LIN {X 0,Y 86.46,Z 826.17,A -85,B 0,C 180,E1 -28946.433,E2 -28946.433} C_VEL
LIN {X 0,Y 94.835,Z 817.694,A -85,B 0,C 180,E1 -28950.553,E2 -28950.553} C_VEL
LIN {X 0,Y 102.155,Z 808.982,A -85,B 0,C 180,E1 -28953.433,E2 -28953.433} C_VEL
LIN {X 0,Y 109.71,Z 798.261,A -85,B 0,C 180,E1 -28955.908,E2 -28955.908} C_VEL
LIN {X 0,Y 115.889,Z 787.44,A -85,B 0,C 180,E1 -28957.648,E2 -28957.648} C_VEL
LIN {X 0,Y 121.383,Z 775.363,A -85,B 0,C 180,E1 -28959.012,E2 -28959.012} C_VEL
LIN {X 0,Y 123.313,Z 770.258,A -85,B 0,C 180,E1 -28959.435,E2 -28959.435} C_VEL
LIN {X 0,Y 124.952,Z 764.764,A -85,B 0,C 180,E1 -28960.101,E2 -28960.101} C_VEL
LIN {X 0,Y 126.471,Z 755.717,A -85,B 0,C 180,E1 -28961.826,E2 -28961.826} C_VEL
LIN {X 0,Y 127.385,Z 746.482,A -85,B 0,C 180,E1 -28963.443,E2 -28963.443} C_VEL
LIN {X 0,Y 127.985,Z 740.687,A -85,B 0,C 180,E1 -28963.94,E2 -28963.94} C_VEL
LIN {X 0,Y 131.877,Z 705.031,A -85,B 0,C 180,E1 -28964.991,E2 -28964.991} C_VEL
LIN {X 0,Y 132.564,Z 694.277,A -85,B 0,C 180,E1 -28966.12,E2 -28966.12} C_VEL
LIN {X 0,Y 131.059,Z 690.593,A -85,B 0,C 180,E1 -28970.158,E2 -28970.158} C_VEL
LIN {X 0,Y 129.868,Z 687.923,A -85,B 0,C 180,E1 -28975.344,E2 -28975.344} C_VEL
LIN {X 0,Y 129.584,Z 687.04,A -85,B 0,C 180,E1 -28978.446,E2 -28978.446} C_VEL
LIN {X 0,Y 129.581,Z 688.078,A -85,B 0,C 180,E1 -28983.109,E2 -28983.109} C_VEL
LIN {X 0,Y 130.12,Z 690.292,A -85,B 0,C 180,E1 -28987.175,E2 -28987.175} C_VEL
LIN {X 0,Y 131.254,Z 694.381,A -85,B 0,C 180,E1 -28991.584,E2 -28991.584} C_VEL
LIN {X 0,Y 132.585,Z 699.79,A -85,B 0,C 180,E1 -28995.273,E2 -28995.273} C_VEL
LIN {X 0,Y 129.78,Z 725.663,A -85,B 0,C 180,E1 -28996.051,E2 -28996.051} C_VEL
LIN {X 0,Y 127.305,Z 745.814,A -85,B 0,C 180,E1 -28996.653,E2 -28996.653} C_VEL
LIN {X 0,Y 124.21,Z 759.298,A -85,B 0,C 180,E1 -28997.284,E2 -28997.284} C_VEL
LIN {X 0,Y 120.227,Z 771.36,A -85,B 0,C 180,E1 -28998.205,E2 -28998.205} C_VEL
LIN {X 0,Y 115.453,Z 782.235,A -85,B 0,C 180,E1 -28999.34,E2 -28999.34} C_VEL
LIN {X 0,Y 109.154,Z 793.548,A -85,B 0,C 180,E1 -29000.991,E2 -29000.991} C_VEL
LIN {X 0,Y 102.148,Z 803.754,A -85,B 0,C 180,E1 -29003.034,E2 -29003.034} C_VEL
LIN {X 0,Y 95.328,Z 812.1,A -85,B 0,C 180,E1 -29005.422,E2 -29005.422} C_VEL
LIN {X 0,Y 87.086,Z 820.636,A -85,B 0,C 180,E1 -29008.961,E2 -29008.961} C_VEL
LIN {X 0,Y 78.237,Z 828.356,A -85,B 0,C 180,E1 -29013.8,E2 -29013.8} C_VEL
LIN {X 0,Y 69.093,Z 834.993,A -85,B 0,C 180,E1 -29020.274,E2 -29020.274} C_VEL
LIN {X 0,Y 62.144,Z 839.341,A -85,B 0,C 180,E1 -29027.262,E2 -29027.262} C_VEL
LIN {X 0,Y 58.152,Z 841.624,A -85,B 0,C 180,E1 -29032.817,E2 -29032.817} C_VEL
LIN {X 0,Y 54.742,Z 843.484,A -85,B 0,C 180,E1 -29039.094,E2 -29039.094} C_VEL
LIN {X 0,Y 52.001,Z 844.896,A -85,B 0,C 180,E1 -29046.074,E2 -29046.074} C_VEL
LIN {X 0,Y 48.874,Z 846.492,A -85,B 0,C 180,E1 -29061.726,E2 -29061.726} C_VEL
LIN {X 0,Y 48.51,Z 846.718,A -85,B 0,C 180,E1 -29069.993,E2 -29069.993} C_VEL
LIN {X 0,Y 48.829,Z 846.519,A -85,B 0,C 180,E1 -29078.268,E2 -29078.268} C_VEL
LIN {X 0,Y 50.012,Z 845.929,A -85,B 0,C 180,E1 -29086.316,E2 -29086.316} C_VEL
LIN {X 0,Y 51.995,Z 844.956,A -85,B 0,C 180,E1 -29093.915,E2 -29093.915} C_VEL
LIN {X 0,Y 54.73,Z 843.578,A -85,B 0,C 180,E1 -29100.9,E2 -29100.9} C_VEL
LIN {X 0,Y 60.066,Z 840.685,A -85,B 0,C 180,E1 -29110.047,E2 -29110.047} C_VEL
LIN {X 0,Y 66.591,Z 836.748,A -85,B 0,C 180,E1 -29117.619,E2 -29117.619} C_VEL
LIN {X 0,Y 74.148,Z 831.639,A -85,B 0,C 180,E1 -29123.665,E2 -29123.665} C_VEL
LIN {X 0,Y 82.281,Z 825.202,A -85,B 0,C 180,E1 -29128.656,E2 -29128.656} C_VEL
LIN {X 0,Y 84.018,Z 823.562,A -85,B 0,C 180,E1 -29129.874,E2 -29129.874} C_VEL
LIN {X 0,Y 78.219,Z 822.134,A -85,B 0,C 180,E1 -29144.362,E2 -29144.362} C_VEL
LIN {X 0,Y 78.822,Z 819.937,A -85,B 0,C 180,E1 -29160,E2 -29160} C_VEL
LIN {X 0,Y 85.752,Z 816.801,A -85,B 0,C 180,E1 -29174.233,E2 -29174.233} C_VEL
LIN {X 0,Y 94.96,Z 813.582,A -85,B 0,C 180,E1 -29183.594,E2 -29183.594} C_VEL
LIN {X 0,Y 94.804,Z 814.301,A -85,B 0,C 180,E1 -29184.407,E2 -29184.407} C_VEL
LIN {X 0,Y 87.113,Z 822.244,A -85,B 0,C 180,E1 -29187.456,E2 -29187.456} C_VEL
LIN {X 0,Y 78.562,Z 829.753,A -85,B 0,C 180,E1 -29191.814,E2 -29191.814} C_VEL
LIN {X 0,Y 70.637,Z 835.789,A -85,B 0,C 180,E1 -29197.263,E2 -29197.263} C_VEL
LIN {X 0,Y 63.363,Z 840.558,A -85,B 0,C 180,E1 -29203.875,E2 -29203.875} C_VEL
LIN {X 0,Y 57.146,Z 844.205,A -85,B 0,C 180,E1 -29212.062,E2 -29212.062} C_VEL
LIN {X 0,Y 53.773,Z 846.089,A -85,B 0,C 180,E1 -29218.488,E2 -29218.488} C_VEL
LIN {X 0,Y 51.191,Z 847.509,A -85,B 0,C 180,E1 -29225.685,E2 -29225.685} C_VEL
LIN {X 0,Y 48.553,Z 849.137,A -85,B 0,C 180,E1 -29241.684,E2 -29241.684} C_VEL
LIN {X 0,Y 48.502,Z 849.357,A -85,B 0,C 180,E1 -29250.007,E2 -29250.007} C_VEL
LIN {X 0,Y 48.555,Z 849.116,A -85,B 0,C 180,E1 -29258.329,E2 -29258.329} C_VEL
LIN {X 0,Y 51.19,Z 847.46,A -85,B 0,C 180,E1 -29274.329,E2 -29274.329} C_VEL
LIN {X 0,Y 53.765,Z 846.011,A -85,B 0,C 180,E1 -29281.531,E2 -29281.531} C_VEL
LIN {X 0,Y 59.08,Z 843.026,A -85,B 0,C 180,E1 -29290.871,E2 -29290.871} C_VEL
LIN {X 0,Y 65.662,Z 838.985,A -85,B 0,C 180,E1 -29298.53,E2 -29298.53} C_VEL
LIN {X 0,Y 73.734,Z 833.34,A -85,B 0,C 180,E1 -29305.118,E2 -29305.118} C_VEL
LIN {X 0,Y 82.731,Z 825.978,A -85,B 0,C 180,E1 -29310.551,E2 -29310.551} C_VEL
LIN {X 0,Y 91.551,Z 817.503,A -85,B 0,C 180,E1 -29314.429,E2 -29314.429} C_VEL
LIN {X 0,Y 99.175,Z 808.792,A -85,B 0,C 180,E1 -29317.114,E2 -29317.114} C_VEL
LIN {X 0,Y 107.013,Z 798.075,A -85,B 0,C 180,E1 -29319.374,E2 -29319.374} C_VEL
LIN {X 0,Y 113.383,Z 787.257,A -85,B 0,C 180,E1 -29320.962,E2 -29320.962} C_VEL
LIN {X 0,Y 119.028,Z 775.186,A -85,B 0,C 180,E1 -29322.201,E2 -29322.201} C_VEL
LIN {X 0,Y 123.519,Z 762.455,A -85,B 0,C 180,E1 -29323.064,E2 -29323.064} C_VEL
LIN {X 0,Y 126.616,Z 749.727,A -85,B 0,C 180,E1 -29323.597,E2 -29323.597} C_VEL
LIN {X 0,Y 127.985,Z 740.687,A -85,B 0,C 180,E1 -29323.94,E2 -29323.94} C_VEL
LIN {X 0,Y 128.477,Z 734.891,A -85,B 0,C 180,E1 -29324.411,E2 -29324.411} C_VEL
LIN {X 0,Y 129.14,Z 716.204,A -85,B 0,C 180,E1 -29327.354,E2 -29327.354} C_VEL
LIN {X 0,Y 129.631,Z 710.401,A -85,B 0,C 180,E1 -29327.808,E2 -29327.808} C_VEL
LIN {X 0,Y 130.259,Z 704.044,A -85,B 0,C 180,E1 -29328.159,E2 -29328.159} C_VEL
LIN {X 0,Y 130.607,Z 699.268,A -85,B 0,C 180,E1 -29328.692,E2 -29328.692} C_VEL
LIN {X 0,Y 129.778,Z 697.071,A -85,B 0,C 180,E1 -29331.436,E2 -29331.436} C_VEL
LIN {X 0,Y 128.943,Z 694.914,A -85,B 0,C 180,E1 -29335.702,E2 -29335.702} C_VEL
LIN {X 0,Y 128.714,Z 694.127,A -85,B 0,C 180,E1 -29338.436,E2 -29338.436} C_VEL
LIN {X 0,Y 128.669,Z 695.009,A -85,B 0,C 180,E1 -29342.563,E2 -29342.563} C_VEL
LIN {X 0,Y 129.078,Z 697.136,A -85,B 0,C 180,E1 -29346.44,E2 -29346.44} C_VEL
LIN {X 0,Y 129.961,Z 700.948,A -85,B 0,C 180,E1 -29350.516,E2 -29350.516} C_VEL
LIN {X 0,Y 130.496,Z 703.71,A -85,B 0,C 180,E1 -29352.441,E2 -29352.441} C_VEL
LIN {X 0,Y 125.582,Z 745.27,A -85,B 0,C 180,E1 -29353.527,E2 -29353.527} C_VEL
LIN {X 0,Y 122.71,Z 758.014,A -85,B 0,C 180,E1 -29354.047,E2 -29354.047} C_VEL
LIN {X 0,Y 118.615,Z 770.448,A -85,B 0,C 180,E1 -29354.859,E2 -29354.859} C_VEL
LIN {X 0,Y 113.301,Z 782.417,A -85,B 0,C 180,E1 -29355.952,E2 -29355.952} C_VEL
LIN {X 0,Y 106.824,Z 793.734,A -85,B 0,C 180,E1 -29357.445,E2 -29357.445} C_VEL
LIN {X 0,Y 99.59,Z 803.943,A -85,B 0,C 180,E1 -29359.282,E2 -29359.282} C_VEL
LIN {X 0,Y 92.501,Z 812.291,A -85,B 0,C 180,E1 -29361.444,E2 -29361.444} C_VEL
LIN {X 0,Y 84.831,Z 819.972,A -85,B 0,C 180,E1 -29364.304,E2 -29364.304} C_VEL
LIN {X 0,Y 75.941,Z 827.453,A -85,B 0,C 180,E1 -29368.449,E2 -29368.449} C_VEL
LIN {X 0,Y 67.442,Z 833.459,A -85,B 0,C 180,E1 -29373.516,E2 -29373.516} C_VEL
LIN {X 0,Y 59.557,Z 838.201,A -85,B 0,C 180,E1 -29379.904,E2 -29379.904} C_VEL
LIN {X 0,Y 52.675,Z 841.817,A -85,B 0,C 180,E1 -29388.148,E2 -29388.148} C_VEL
LIN {X 0,Y 48.78,Z 843.677,A -85,B 0,C 180,E1 -29394.801,E2 -29394.801} C_VEL
LIN {X 0,Y 45.601,Z 845.089,A -85,B 0,C 180,E1 -29402.453,E2 -29402.453} C_VEL
LIN {X 0,Y 41.877,Z 846.685,A -85,B 0,C 180,E1 -29420.331,E2 -29420.331} C_VEL
LIN {X 0,Y 41.428,Z 846.911,A -85,B 0,C 180,E1 -29429.992,E2 -29429.992} C_VEL
LIN {X 0,Y 41.826,Z 846.712,A -85,B 0,C 180,E1 -29439.665,E2 -29439.665} C_VEL
LIN {X 0,Y 45.594,Z 845.149,A -85,B 0,C 180,E1 -29457.535,E2 -29457.535} C_VEL
LIN {X 0,Y 48.767,Z 843.771,A -85,B 0,C 180,E1 -29465.193,E2 -29465.193} C_VEL
LIN {X 0,Y 54.802,Z 840.878,A -85,B 0,C 180,E1 -29474.848,E2 -29474.848} C_VEL
LIN {X 0,Y 62.034,Z 836.939,A -85,B 0,C 180,E1 -29482.462,E2 -29482.462} C_VEL
LIN {X 0,Y 70.178,Z 831.829,A -85,B 0,C 180,E1 -29488.336,E2 -29488.336} C_VEL
LIN {X 0,Y 75.329,Z 828.108,A -85,B 0,C 180,E1 -29491.331,E2 -29491.331} C_VEL
LIN {X 0,Y 76.161,Z 827.21,A -85,B 0,C 180,E1 -29492.522,E2 -29492.522} C_VEL
LIN {X 0,Y 71.978,Z 825.743,A -85,B 0,C 180,E1 -29508.738,E2 -29508.738} C_VEL
LIN {X 0,Y 74.833,Z 823.501,A -85,B 0,C 180,E1 -29525.389,E2 -29525.389} C_VEL
LIN {X 0,Y 85.395,Z 819.982,A -85,B 0,C 180,E1 -29540.986,E2 -29540.986} C_VEL
LIN {X 0,Y 86.136,Z 819.753,A -85,B 0,C 180,E1 -29541.678,E2 -29541.678} C_VEL
LIN {X 0,Y 84.717,Z 821.456,A -85,B 0,C 180,E1 -29542.901,E2 -29542.901} C_VEL
LIN {X 0,Y 75.043,Z 829.563,A -85,B 0,C 180,E1 -29547.176,E2 -29547.176} C_VEL
LIN {X 0,Y 66.551,Z 835.598,A -85,B 0,C 180,E1 -29552.357,E2 -29552.357} C_VEL
LIN {X 0,Y 58.639,Z 840.366,A -85,B 0,C 180,E1 -29558.837,E2 -29558.837} C_VEL
LIN {X 0,Y 51.721,Z 844.013,A -85,B 0,C 180,E1 -29567.212,E2 -29567.212} C_VEL
LIN {X 0,Y 47.83,Z 845.896,A -85,B 0,C 180,E1 -29574.012,E2 -29574.012} C_VEL
LIN {X 0,Y 44.782,Z 847.316,A -85,B 0,C 180,E1 -29581.922,E2 -29581.922} C_VEL
LIN {X 0,Y 41.528,Z 848.944,A -85,B 0,C 180,E1 -29600.265,E2 -29600.265} C_VEL
LIN {X 0,Y 41.412,Z 849.164,A -85,B 0,C 180,E1 -29610.008,E2 -29610.008} C_VEL
LIN {X 0,Y 41.529,Z 848.923,A -85,B 0,C 180,E1 -29619.751,E2 -29619.751} C_VEL
LIN {X 0,Y 44.782,Z 847.266,A -85,B 0,C 180,E1 -29638.095,E2 -29638.095} C_VEL
LIN {X 0,Y 47.823,Z 845.817,A -85,B 0,C 180,E1 -29646.011,E2 -29646.011} C_VEL
LIN {X 0,Y 53.889,Z 842.832,A -85,B 0,C 180,E1 -29655.839,E2 -29655.839} C_VEL
LIN {X 0,Y 61.185,Z 838.791,A -85,B 0,C 180,E1 -29663.526,E2 -29663.526} C_VEL
LIN {X 0,Y 70.675,Z 832.593,A -85,B 0,C 180,E1 -29670.406,E2 -29670.406} C_VEL
LIN {X 0,Y 79.474,Z 825.785,A -85,B 0,C 180,E1 -29675.024,E2 -29675.024} C_VEL
LIN {X 0,Y 88.709,Z 817.312,A -85,B 0,C 180,E1 -29678.583,E2 -29678.583} C_VEL
LIN {X 0,Y 96.629,Z 808.603,A -85,B 0,C 180,E1 -29681.007,E2 -29681.007} C_VEL
LIN {X 0,Y 104.727,Z 797.888,A -85,B 0,C 180,E1 -29683.004,E2 -29683.004} C_VEL
LIN {X 0,Y 111.273,Z 787.074,A -85,B 0,C 180,E1 -29684.414,E2 -29684.414} C_VEL
LIN {X 0,Y 117.056,Z 775.009,A -85,B 0,C 180,E1 -29685.506,E2 -29685.506} C_VEL
LIN {X 0,Y 121.644,Z 762.29,A -85,B 0,C 180,E1 -29686.258,E2 -29686.258} C_VEL
LIN {X 0,Y 124.881,Z 749.158,A -85,B 0,C 180,E1 -29686.738,E2 -29686.738} C_VEL
LIN {X 0,Y 127.205,Z 731.857,A -85,B 0,C 180,E1 -29687.264,E2 -29687.264} C_VEL
LIN {X 0,Y 129.631,Z 710.401,A -85,B 0,C 180,E1 -29687.808,E2 -29687.808} C_VEL
LIN {X 0,Y 129.736,Z 707.831,A -85,B 0,C 180,E1 -29688.259,E2 -29688.259} C_VEL
LIN {X 0,Y 129.517,Z 705.447,A -85,B 0,C 180,E1 -29689.408,E2 -29689.408} C_VEL
LIN {X 0,Y 129.091,Z 703.798,A -85,B 0,C 180,E1 -29691.014,E2 -29691.014} C_VEL
LIN {X 0,Y 128.425,Z 702.558,A -85,B 0,C 180,E1 -29693.701,E2 -29693.701} C_VEL
LIN {X 0,Y 127.977,Z 701.798,A -85,B 0,C 180,E1 -29696.453,E2 -29696.453} C_VEL
LIN {X 0,Y 127.848,Z 701.182,A -85,B 0,C 180,E1 -29698.425,E2 -29698.425} C_VEL
LIN {X 0,Y 127.78,Z 702.05,A -85,B 0,C 180,E1 -29702.295,E2 -29702.295} C_VEL
LIN {X 0,Y 128.083,Z 704.162,A -85,B 0,C 180,E1 -29705.905,E2 -29705.905} C_VEL
LIN {X 0,Y 128.712,Z 707.544,A -85,B 0,C 180,E1 -29709.428,E2 -29709.428} C_VEL
LIN {X 0,Y 124.023,Z 745.927,A -85,B 0,C 180,E1 -29710.359,E2 -29710.359} C_VEL
LIN {X 0,Y 120.97,Z 758.904,A -85,B 0,C 180,E1 -29710.815,E2 -29710.815} C_VEL
LIN {X 0,Y 116.583,Z 771.711,A -85,B 0,C 180,E1 -29711.582,E2 -29711.582} C_VEL
LIN {X 0,Y 111.562,Z 782.599,A -85,B 0,C 180,E1 -29712.451,E2 -29712.451} C_VEL
LIN {X 0,Y 104.92,Z 793.92,A -85,B 0,C 180,E1 -29713.756,E2 -29713.756} C_VEL
LIN {X 0,Y 97.481,Z 804.13,A -85,B 0,C 180,E1 -29715.35,E2 -29715.35} C_VEL
LIN {X 0,Y 90.145,Z 812.481,A -85,B 0,C 180,E1 -29717.234,E2 -29717.234} C_VEL
LIN {X 0,Y 82.166,Z 820.163,A -85,B 0,C 180,E1 -29719.791,E2 -29719.791} C_VEL
LIN {X 0,Y 72.817,Z 827.646,A -85,B 0,C 180,E1 -29723.514,E2 -29723.514} C_VEL
LIN {X 0,Y 63.8,Z 833.652,A -85,B 0,C 180,E1 -29728.197,E2 -29728.197} C_VEL
LIN {X 0,Y 55.274,Z 838.394,A -85,B 0,C 180,E1 -29734.254,E2 -29734.254} C_VEL
LIN {X 0,Y 47.629,Z 842.01,A -85,B 0,C 180,E1 -29742.448,E2 -29742.448} C_VEL
LIN {X 0,Y 43.172,Z 843.871,A -85,B 0,C 180,E1 -29749.362,E2 -29749.362} C_VEL
LIN {X 0,Y 39.449,Z 845.282,A -85,B 0,C 180,E1 -29757.683,E2 -29757.683} C_VEL
LIN {X 0,Y 34.892,Z 846.878,A -85,B 0,C 180,E1 -29778.37,E2 -29778.37} C_VEL
LIN {X 0,Y 34.331,Z 847.104,A -85,B 0,C 180,E1 -29789.99,E2 -29789.99} C_VEL
LIN {X 0,Y 34.843,Z 846.905,A -85,B 0,C 180,E1 -29801.627,E2 -29801.627} C_VEL
LIN {X 0,Y 39.441,Z 845.341,A -85,B 0,C 180,E1 -29822.304,E2 -29822.304} C_VEL
LIN {X 0,Y 43.159,Z 843.963,A -85,B 0,C 180,E1 -29830.634,E2 -29830.634} C_VEL
LIN {X 0,Y 50.007,Z 841.07,A -85,B 0,C 180,E1 -29840.61,E2 -29840.61} C_VEL
LIN {X 0,Y 57.989,Z 837.129,A -85,B 0,C 180,E1 -29848.022,E2 -29848.022} C_VEL
LIN {X 0,Y 66.375,Z 832.252,A -85,B 0,C 180,E1 -29853.334,E2 -29853.334} C_VEL
LIN {X 0,Y 68.453,Z 830.543,A -85,B 0,C 180,E1 -29855.752,E2 -29855.752} C_VEL
LIN {X 0,Y 66.127,Z 829.096,A -85,B 0,C 180,E1 -29873.899,E2 -29873.899} C_VEL
LIN {X 0,Y 71.877,Z 826.736,A -85,B 0,C 180,E1 -29892.128,E2 -29892.128} C_VEL
LIN {X 0,Y 76.932,Z 825.362,A -85,B 0,C 180,E1 -29899.207,E2 -29899.207} C_VEL
LIN {X 0,Y 75.181,Z 827.044,A -85,B 0,C 180,E1 -29900.816,E2 -29900.816} C_VEL
LIN {X 0,Y 65.075,Z 834.136,A -85,B 0,C 180,E1 -29905.594,E2 -29905.594} C_VEL
LIN {X 0,Y 57.252,Z 838.74,A -85,B 0,C 180,E1 -29910.776,E2 -29910.776} C_VEL
LIN {X 0,Y 49.201,Z 842.747,A -85,B 0,C 180,E1 -29918.233,E2 -29918.233} C_VEL
LIN {X 0,Y 42.262,Z 845.703,A -85,B 0,C 180,E1 -29928.316,E2 -29928.316} C_VEL
LIN {X 0,Y 38.637,Z 847.122,A -85,B 0,C 180,E1 -29936.939,E2 -29936.939} C_VEL
LIN {X 0,Y 34.531,Z 848.75,A -85,B 0,C 180,E1 -29958.267,E2 -29958.267} C_VEL
LIN {X 0,Y 34.307,Z 848.971,A -85,B 0,C 180,E1 -29970.01,E2 -29970.01} C_VEL
LIN {X 0,Y 34.533,Z 848.729,A -85,B 0,C 180,E1 -29981.752,E2 -29981.752} C_VEL
LIN {X 0,Y 38.638,Z 847.071,A -85,B 0,C 180,E1 -30003.081,E2 -30003.081} C_VEL
LIN {X 0,Y 42.257,Z 845.622,A -85,B 0,C 180,E1 -30011.712,E2 -30011.712} C_VEL
LIN {X 0,Y 49.189,Z 842.638,A -85,B 0,C 180,E1 -30021.807,E2 -30021.807} C_VEL
LIN {X 0,Y 57.243,Z 838.598,A -85,B 0,C 180,E1 -30029.261,E2 -30029.261} C_VEL
LIN {X 0,Y 66.193,Z 833.231,A -85,B 0,C 180,E1 -30035.014,E2 -30035.014} C_VEL
LIN {X 0,Y 75.158,Z 826.814,A -85,B 0,C 180,E1 -30039.253,E2 -30039.253} C_VEL
LIN {X 0,Y 84.746,Z 818.677,A -85,B 0,C 180,E1 -30042.507,E2 -30042.507} C_VEL
LIN {X 0,Y 92.912,Z 810.333,A -85,B 0,C 180,E1 -30044.683,E2 -30044.683} C_VEL
LIN {X 0,Y 101.204,Z 800.015,A -85,B 0,C 180,E1 -30046.472,E2 -30046.472} C_VEL
LIN {X 0,Y 108.738,Z 788.416,A -85,B 0,C 180,E1 -30047.85,E2 -30047.85} C_VEL
LIN {X 0,Y 114.635,Z 776.765,A -85,B 0,C 180,E1 -30048.8,E2 -30048.8} C_VEL
LIN {X 0,Y 119.306,Z 764.743,A -85,B 0,C 180,E1 -30049.436,E2 -30049.436} C_VEL
LIN {X 0,Y 122.867,Z 751.939,A -85,B 0,C 180,E1 -30049.855,E2 -30049.855} C_VEL
LIN {X 0,Y 125.197,Z 737.19,A -85,B 0,C 180,E1 -30050.305,E2 -30050.305} C_VEL
LIN {X 0,Y 128.68,Z 707.099,A -85,B 0,C 180,E1 -30051.015,E2 -30051.015} C_VEL
LIN {X 0,Y 128.913,Z 704.421,A -85,B 0,C 180,E1 -30051.298,E2 -30051.298} C_VEL
LIN {X 0,Y 128.031,Z 701.961,A -85,B 0,C 180,E1 -30055.967,E2 -30055.967} C_VEL
LIN {X 0,Y 127.977,Z 701.798,A -85,B 0,C 180,E1 -30056.453,E2 -30056.453} C_VEL
LIN {X 0,Y 127.743,Z 702.175,A -85,B 0,C 180,E1 -30058.174,E2 -30058.174} C_VEL
LIN {X 0,Y 127.477,Z 703.765,A -85,B 0,C 180,E1 -30059.798,E2 -30059.798} C_VEL
LIN {X 0,Y 127.018,Z 710.164,A -85,B 0,C 180,E1 -30064.224,E2 -30064.224} C_VEL
LIN {X 0,Y 127.072,Z 710.961,A -85,B 0,C 180,E1 -30065.091,E2 -30065.091} C_VEL
LIN {X 0,Y 127.212,Z 712.043,A -85,B 0,C 180,E1 -30066.344,E2 -30066.344} C_VEL
LIN {X 0,Y 123.014,Z 745.705,A -85,B 0,C 180,E1 -30067.104,E2 -30067.104} C_VEL
LIN {X 0,Y 119.845,Z 759.068,A -85,B 0,C 180,E1 -30067.494,E2 -30067.494} C_VEL
LIN {X 0,Y 115.371,Z 771.886,A -85,B 0,C 180,E1 -30068.139,E2 -30068.139} C_VEL
LIN {X 0,Y 110.25,Z 782.781,A -85,B 0,C 180,E1 -30068.848,E2 -30068.848} C_VEL
LIN {X 0,Y 103.464,Z 794.105,A -85,B 0,C 180,E1 -30069.943,E2 -30069.943} C_VEL
LIN {X 0,Y 95.848,Z 804.319,A -85,B 0,C 180,E1 -30071.257,E2 -30071.257} C_VEL
LIN {X 0,Y 88.303,Z 812.671,A -85,B 0,C 180,E1 -30072.833,E2 -30072.833} C_VEL
LIN {X 0,Y 78.631,Z 821.506,A -85,B 0,C 180,E1 -30075.402,E2 -30075.402} C_VEL
LIN {X 0,Y 68.694,Z 828.935,A -85,B 0,C 180,E1 -30078.839,E2 -30078.839} C_VEL
LIN {X 0,Y 57.668,Z 835.571,A -85,B 0,C 180,E1 -30083.919,E2 -30083.919} C_VEL
LIN {X 0,Y 48.67,Z 839.922,A -85,B 0,C 180,E1 -30089.944,E2 -30089.944} C_VEL
LIN {X 0,Y 43.149,Z 842.204,A -85,B 0,C 180,E1 -30095.462,E2 -30095.462} C_VEL
LIN {X 0,Y 38.072,Z 844.064,A -85,B 0,C 180,E1 -30102.394,E2 -30102.394} C_VEL
LIN {X 0,Y 33.651,Z 845.476,A -85,B 0,C 180,E1 -30111.192,E2 -30111.192} C_VEL
LIN {X 0,Y 27.969,Z 847.072,A -85,B 0,C 180,E1 -30135.435,E2 -30135.435} C_VEL
LIN {X 0,Y 27.248,Z 847.297,A -85,B 0,C 180,E1 -30149.988,E2 -30149.988} C_VEL
LIN {X 0,Y 27.93,Z 847.097,A -85,B 0,C 180,E1 -30164.561,E2 -30164.561} C_VEL
LIN {X 0,Y 30.175,Z 846.507,A -85,B 0,C 180,E1 -30177.75,E2 -30177.75} C_VEL
LIN {X 0,Y 33.641,Z 845.534,A -85,B 0,C 180,E1 -30188.796,E2 -30188.796} C_VEL
LIN {X 0,Y 38.056,Z 844.155,A -85,B 0,C 180,E1 -30197.607,E2 -30197.607} C_VEL
LIN {X 0,Y 45.824,Z 841.261,A -85,B 0,C 180,E1 -30207.5,E2 -30207.5} C_VEL
LIN {X 0,Y 54.568,Z 837.319,A -85,B 0,C 180,E1 -30214.347,E2 -30214.347} C_VEL
LIN {X 0,Y 60.729,Z 834.03,A -85,B 0,C 180,E1 -30217.775,E2 -30217.775} C_VEL
LIN {X 0,Y 60.894,Z 833.617,A -85,B 0,C 180,E1 -30219.742,E2 -30219.742} C_VEL
LIN {X 0,Y 60.88,Z 832.161,A -85,B 0,C 180,E1 -30240,E2 -30240} C_VEL
LIN {X 0,Y 67.672,Z 830.257,A -85,B 0,C 180,E1 -30256.159,E2 -30256.159} C_VEL
LIN {X 0,Y 66.467,Z 831.366,A -85,B 0,C 180,E1 -30257.913,E2 -30257.913} C_VEL
LIN {X 0,Y 57.026,Z 836.945,A -85,B 0,C 180,E1 -30262.453,E2 -30262.453} C_VEL
LIN {X 0,Y 47.983,Z 841.319,A -85,B 0,C 180,E1 -30268.518,E2 -30268.518} C_VEL
LIN {X 0,Y 42.382,Z 843.628,A -85,B 0,C 180,E1 -30274.006,E2 -30274.006} C_VEL
LIN {X 0,Y 37.237,Z 845.509,A -85,B 0,C 180,E1 -30280.993,E2 -30280.993} C_VEL
LIN {X 0,Y 32.898,Z 846.929,A -85,B 0,C 180,E1 -30290.156,E2 -30290.156} C_VEL
LIN {X 0,Y 27.612,Z 848.557,A -85,B 0,C 180,E1 -30315.267,E2 -30315.267} C_VEL
LIN {X 0,Y 27.218,Z 848.778,A -85,B 0,C 180,E1 -30330.012,E2 -30330.012} C_VEL
LIN {X 0,Y 27.614,Z 848.535,A -85,B 0,C 180,E1 -30344.757,E2 -30344.757} C_VEL
LIN {X 0,Y 32.9,Z 846.878,A -85,B 0,C 180,E1 -30369.868,E2 -30369.868} C_VEL
LIN {X 0,Y 37.231,Z 845.428,A -85,B 0,C 180,E1 -30379.043,E2 -30379.043} C_VEL
LIN {X 0,Y 45.13,Z 842.443,A -85,B 0,C 180,E1 -30388.94,E2 -30388.94} C_VEL
LIN {X 0,Y 53.954,Z 838.404,A -85,B 0,C 180,E1 -30395.771,E2 -30395.771} C_VEL
LIN {X 0,Y 64.709,Z 832.281,A -85,B 0,C 180,E1 -30401.386,E2 -30401.386} C_VEL
LIN {X 0,Y 74.582,Z 825.4,A -85,B 0,C 180,E1 -30405.003,E2 -30405.003} C_VEL
LIN {X 0,Y 84.554,Z 816.93,A -85,B 0,C 180,E1 -30407.605,E2 -30407.605} C_VEL
LIN {X 0,Y 92.976,Z 808.224,A -85,B 0,C 180,E1 -30409.33,E2 -30409.33} C_VEL
LIN {X 0,Y 101.492,Z 797.516,A -85,B 0,C 180,E1 -30410.685,E2 -30410.685} C_VEL
LIN {X 0,Y 108.329,Z 786.709,A -85,B 0,C 180,E1 -30411.653,E2 -30411.653} C_VEL
LIN {X 0,Y 114.332,Z 774.654,A -85,B 0,C 180,E1 -30412.41,E2 -30412.41} C_VEL
LIN {X 0,Y 119.074,Z 761.958,A -85,B 0,C 180,E1 -30412.906,E2 -30412.906} C_VEL
LIN {X 0,Y 122.47,Z 748.533,A -85,B 0,C 180,E1 -30413.24,E2 -30413.24} C_VEL
LIN {X 0,Y 124.846,Z 731.669,A -85,B 0,C 180,E1 -30413.625,E2 -30413.625} C_VEL
LIN {X 0,Y 127.405,Z 709.97,A -85,B 0,C 180,E1 -30414.133,E2 -30414.133} C_VEL
LIN {X 0,Y 126.974,Z 708.299,A -85,B 0,C 180,E1 -30418.414,E2 -30418.414} C_VEL
LIN {X 0,Y 126.884,Z 708.928,A -85,B 0,C 180,E1 -30421.587,E2 -30421.587} C_VEL
LIN {X 0,Y 127.039,Z 710.648,A -85,B 0,C 180,E1 -30424.701,E2 -30424.701} C_VEL
LIN {X 0,Y 127.072,Z 710.961,A -85,B 0,C 180,E1 -30425.091,E2 -30425.091} C_VEL
LIN {X 0,Y 127.037,Z 712.212,A -85,B 0,C 180,E1 -30425.671,E2 -30425.671} C_VEL
LIN {X 0,Y 126.791,Z 714.634,A -85,B 0,C 180,E1 -30425.91,E2 -30425.91} C_VEL
LIN {X 0,Y 126.263,Z 718.398,A -85,B 0,C 180,E1 -30425.62,E2 -30425.62} C_VEL
LIN {X 0,Y 124.887,Z 727.073,A -85,B 0,C 180,E1 -30423.906,E2 -30423.906} C_VEL
LIN {X 0,Y 124.355,Z 730.999,A -85,B 0,C 180,E1 -30423.547,E2 -30423.547} C_VEL
LIN {X 0,Y 124.256,Z 731.801,A -85,B 0,C 180,E1 -30423.548,E2 -30423.548} C_VEL
LIN {X 0,Y 121.901,Z 748.043,A -85,B 0,C 180,E1 -30423.868,E2 -30423.868} C_VEL
LIN {X 0,Y 118.476,Z 761.412,A -85,B 0,C 180,E1 -30424.169,E2 -30424.169} C_VEL
LIN {X 0,Y 114.584,Z 772.061,A -85,B 0,C 180,E1 -30424.634,E2 -30424.634} C_VEL
LIN {X 0,Y 109.384,Z 782.963,A -85,B 0,C 180,E1 -30425.175,E2 -30425.175} C_VEL
LIN {X 0,Y 102.479,Z 794.29,A -85,B 0,C 180,E1 -30426.038,E2 -30426.038} C_VEL
LIN {X 0,Y 94.719,Z 804.507,A -85,B 0,C 180,E1 -30427.045,E2 -30427.045} C_VEL
LIN {X 0,Y 87.004,Z 812.861,A -85,B 0,C 180,E1 -30428.276,E2 -30428.276} C_VEL
LIN {X 0,Y 78.498,Z 820.547,A -85,B 0,C 180,E1 -30429.971,E2 -30429.971} C_VEL
LIN {X 0,Y 68.401,Z 828.031,A -85,B 0,C 180,E1 -30432.535,E2 -30432.535} C_VEL
LIN {X 0,Y 58.452,Z 834.037,A -85,B 0,C 180,E1 -30435.854,E2 -30435.854} C_VEL
LIN {X 0,Y 48.706,Z 838.781,A -85,B 0,C 180,E1 -30440.278,E2 -30440.278} C_VEL
LIN {X 0,Y 39.453,Z 842.398,A -85,B 0,C 180,E1 -30447.025,E2 -30447.025} C_VEL
LIN {X 0,Y 33.693,Z 844.257,A -85,B 0,C 180,E1 -30453.434,E2 -30453.434} C_VEL
LIN {X 0,Y 28.464,Z 845.669,A -85,B 0,C 180,E1 -30462.19,E2 -30462.19} C_VEL
LIN {X 0,Y 21.181,Z 847.265,A -85,B 0,C 180,E1 -30490.605,E2 -30490.605} C_VEL
LIN {X 0,Y 20.16,Z 847.49,A -85,B 0,C 180,E1 -30509.983,E2 -30509.983} C_VEL
LIN {X 0,Y 21.15,Z 847.29,A -85,B 0,C 180,E1 -30529.391,E2 -30529.391} C_VEL
LIN {X 0,Y 24.114,Z 846.699,A -85,B 0,C 180,E1 -30545.636,E2 -30545.636} C_VEL
LIN {X 0,Y 28.453,Z 845.727,A -85,B 0,C 180,E1 -30557.799,E2 -30557.799} C_VEL
LIN {X 0,Y 33.676,Z 844.347,A -85,B 0,C 180,E1 -30566.574,E2 -30566.574} C_VEL
LIN {X 0,Y 42.431,Z 841.453,A -85,B 0,C 180,E1 -30575.622,E2 -30575.622} C_VEL
LIN {X 0,Y 53.411,Z 836.765,A -85,B 0,C 180,E1 -30582.174,E2 -30582.174} C_VEL
LIN {X 0,Y 53.691,Z 836.385,A -85,B 0,C 180,E1 -30584.823,E2 -30584.823} C_VEL
LIN {X 0,Y 56.799,Z 834.861,A -85,B 0,C 180,E1 -30608.206,E2 -30608.206} C_VEL
LIN {X 0,Y 58.714,Z 834.619,A -85,B 0,C 180,E1 -30613.851,E2 -30613.851} C_VEL
LIN {X 0,Y 48.201,Z 839.791,A -85,B 0,C 180,E1 -30618.63,E2 -30618.63} C_VEL
LIN {X 0,Y 38.846,Z 843.436,A -85,B 0,C 180,E1 -30625.252,E2 -30625.252} C_VEL
LIN {X 0,Y 32.998,Z 845.316,A -85,B 0,C 180,E1 -30631.598,E2 -30631.598} C_VEL
LIN {X 0,Y 27.797,Z 846.736,A -85,B 0,C 180,E1 -30640.688,E2 -30640.688} C_VEL
LIN {X 0,Y 20.801,Z 848.364,A -85,B 0,C 180,E1 -30670.271,E2 -30670.271} C_VEL
LIN {X 0,Y 20.102,Z 848.584,A -85,B 0,C 180,E1 -30690.017,E2 -30690.017} C_VEL
LIN {X 0,Y 20.805,Z 848.341,A -85,B 0,C 180,E1 -30709.76,E2 -30709.76} C_VEL
LIN {X 0,Y 27.8,Z 846.683,A -85,B 0,C 180,E1 -30739.341,E2 -30739.341} C_VEL
LIN {X 0,Y 32.995,Z 845.233,A -85,B 0,C 180,E1 -30748.448,E2 -30748.448} C_VEL
LIN {X 0,Y 41.899,Z 842.249,A -85,B 0,C 180,E1 -30757.321,E2 -30757.321} C_VEL
LIN {X 0,Y 51.444,Z 838.211,A -85,B 0,C 180,E1 -30763.02,E2 -30763.02} C_VEL
LIN {X 0,Y 62.793,Z 832.086,A -85,B 0,C 180,E1 -30767.584,E2 -30767.584} C_VEL
LIN {X 0,Y 73.061,Z 825.208,A -85,B 0,C 180,E1 -30770.416,E2 -30770.416} C_VEL
LIN {X 0,Y 83.319,Z 816.739,A -85,B 0,C 180,E1 -30772.382,E2 -30772.382} C_VEL
LIN {X 0,Y 91.925,Z 808.034,A -85,B 0,C 180,E1 -30773.689,E2 -30773.689} C_VEL
LIN {X 0,Y 100.587,Z 797.329,A -85,B 0,C 180,E1 -30774.674,E2 -30774.674} C_VEL
LIN {X 0,Y 107.528,Z 786.526,A -85,B 0,C 180,E1 -30775.395,E2 -30775.395} C_VEL
LIN {X 0,Y 113.613,Z 774.477,A -85,B 0,C 180,E1 -30775.956,E2 -30775.956} C_VEL
LIN {X 0,Y 118.408,Z 761.792,A -85,B 0,C 180,E1 -30776.311,E2 -30776.311} C_VEL
LIN {X 0,Y 121.733,Z 748.909,A -85,B 0,C 180,E1 -30776.536,E2 -30776.536} C_VEL
LIN {X 0,Y 124.097,Z 732.894,A -85,B 0,C 180,E1 -30776.855,E2 -30776.855} C_VEL
LIN {X 0,Y 126.161,Z 715.782,A -85,B 0,C 180,E1 -30777.206,E2 -30777.206} C_VEL
LIN {X 0,Y 126.098,Z 715.431,A -85,B 0,C 180,E1 -30778.403,E2 -30778.403} C_VEL
LIN {X 0,Y 126.008,Z 715.803,A -85,B 0,C 180,E1 -30780.877,E2 -30780.877} C_VEL
LIN {X 0,Y 126.042,Z 717.014,A -85,B 0,C 180,E1 -30783.286,E2 -30783.286} C_VEL
LIN {X 0,Y 124.256,Z 731.801,A -85,B 0,C 180,E1 -30783.548,E2 -30783.548} C_VEL
LIN {X 0,Y 123.512,Z 737.653,A -85,B 0,C 180,E1 -30783.329,E2 -30783.329} C_VEL
LIN {X 0,Y 121.914,Z 747.116,A -85,B 0,C 180,E1 -30782.106,E2 -30782.106} C_VEL
LIN {X 0,Y 119.712,Z 756.449,A -85,B 0,C 180,E1 -30780.919,E2 -30780.919} C_VEL
LIN {X 0,Y 118.009,Z 762.087,A -85,B 0,C 180,E1 -30780.748,E2 -30780.748} C_VEL
LIN {X 0,Y 113.344,Z 774.239,A -85,B 0,C 180,E1 -30781.14,E2 -30781.14} C_VEL
LIN {X 0,Y 108.099,Z 784.685,A -85,B 0,C 180,E1 -30781.547,E2 -30781.547} C_VEL
LIN {X 0,Y 101.102,Z 795.739,A -85,B 0,C 180,E1 -30782.137,E2 -30782.137} C_VEL
LIN {X 0,Y 93.241,Z 805.721,A -85,B 0,C 180,E1 -30782.852,E2 -30782.852} C_VEL
LIN {X 0,Y 84.529,Z 814.689,A -85,B 0,C 180,E1 -30783.822,E2 -30783.822} C_VEL
LIN {X 0,Y 74.503,Z 823.115,A -85,B 0,C 180,E1 -30785.292,E2 -30785.292} C_VEL
LIN {X 0,Y 63.776,Z 830.402,A -85,B 0,C 180,E1 -30787.316,E2 -30787.316} C_VEL
LIN {X 0,Y 53.506,Z 835.958,A -85,B 0,C 180,E1 -30789.863,E2 -30789.863} C_VEL
LIN {X 0,Y 43.358,Z 840.309,A -85,B 0,C 180,E1 -30793.424,E2 -30793.424} C_VEL
LIN {X 0,Y 36.768,Z 842.592,A -85,B 0,C 180,E1 -30797.085,E2 -30797.085} C_VEL
LIN {X 0,Y 30.357,Z 844.451,A -85,B 0,C 180,E1 -30802.148,E2 -30802.148} C_VEL
LIN {X 0,Y 24.273,Z 845.863,A -85,B 0,C 180,E1 -30809.677,E2 -30809.677} C_VEL
LIN {X 0,Y 14.692,Z 847.458,A -85,B 0,C 180,E1 -30841.397,E2 -30841.397} C_VEL
LIN {X 0,Y 13.06,Z 847.683,A -85,B 0,C 180,E1 -30869.974,E2 -30869.974} C_VEL
LIN {X 0,Y 14.647,Z 847.483,A -85,B 0,C 180,E1 -30898.647,E2 -30898.647} C_VEL
LIN {X 0,Y 18.808,Z 846.892,A -85,B 0,C 180,E1 -30918.333,E2 -30918.333} C_VEL
LIN {X 0,Y 24.262,Z 845.919,A -85,B 0,C 180,E1 -30930.316,E2 -30930.316} C_VEL
LIN {X 0,Y 30.34,Z 844.54,A -85,B 0,C 180,E1 -30937.875,E2 -30937.875} C_VEL
LIN {X 0,Y 40.018,Z 841.645,A -85,B 0,C 180,E1 -30944.96,E2 -30944.96} C_VEL
LIN {X 0,Y 45.391,Z 839.657,A -85,B 0,C 180,E1 -30947.506,E2 -30947.506} C_VEL
LIN {X 0,Y 46.969,Z 838.937,A -85,B 0,C 180,E1 -30949.668,E2 -30949.668} C_VEL
LIN {X 0,Y 49.877,Z 838.058,A -85,B 0,C 180,E1 -30968.1,E2 -30968.1} C_VEL
LIN {X 0,Y 49.822,Z 838.166,A -85,B 0,C 180,E1 -30969.14,E2 -30969.14} C_VEL
LIN {X 0,Y 39.697,Z 842.17,A -85,B 0,C 180,E1 -30973.203,E2 -30973.203} C_VEL
LIN {X 0,Y 29.885,Z 845.123,A -85,B 0,C 180,E1 -30979.871,E2 -30979.871} C_VEL
LIN {X 0,Y 23.763,Z 846.542,A -85,B 0,C 180,E1 -30987.5,E2 -30987.5} C_VEL
LIN {X 0,Y 14.29,Z 848.17,A -85,B 0,C 180,E1 -31020.568,E2 -31020.568} C_VEL
LIN {X 0,Y 12.991,Z 848.391,A -85,B 0,C 180,E1 -31050.026,E2 -31050.026} C_VEL
LIN {X 0,Y 14.295,Z 848.147,A -85,B 0,C 180,E1 -31079.474,E2 -31079.474} C_VEL
LIN {X 0,Y 23.769,Z 846.488,A -85,B 0,C 180,E1 -31112.534,E2 -31112.534} C_VEL
LIN {X 0,Y 29.888,Z 845.039,A -85,B 0,C 180,E1 -31120.181,E2 -31120.181} C_VEL
LIN {X 0,Y 39.699,Z 842.055,A -85,B 0,C 180,E1 -31126.856,E2 -31126.856} C_VEL
LIN {X 0,Y 52.221,Z 836.887,A -85,B 0,C 180,E1 -31131.661,E2 -31131.661} C_VEL
LIN {X 0,Y 63.549,Z 830.787,A -85,B 0,C 180,E1 -31134.505,E2 -31134.505} C_VEL
LIN {X 0,Y 73.958,Z 823.726,A -85,B 0,C 180,E1 -31136.233,E2 -31136.233} C_VEL
LIN {X 0,Y 84.424,Z 814.941,A -85,B 0,C 180,E1 -31137.453,E2 -31137.453} C_VEL
LIN {X 0,Y 93.17,Z 805.92,A -85,B 0,C 180,E1 -31138.235,E2 -31138.235} C_VEL
LIN {X 0,Y 101.054,Z 795.893,A -85,B 0,C 180,E1 -31138.8,E2 -31138.8} C_VEL
LIN {X 0,Y 108.069,Z 784.797,A -85,B 0,C 180,E1 -31139.237,E2 -31139.237} C_VEL
LIN {X 0,Y 113.334,Z 774.3,A -85,B 0,C 180,E1 -31139.532,E2 -31139.532} C_VEL
LIN {X 0,Y 117.724,Z 762.983,A -85,B 0,C 180,E1 -31139.718,E2 -31139.718} C_VEL
LIN {X 0,Y 121.315,Z 749.714,A -85,B 0,C 180,E1 -31139.868,E2 -31139.868} C_VEL
LIN {X 0,Y 123.732,Z 734.246,A -85,B 0,C 180,E1 -31140.133,E2 -31140.133} C_VEL
LIN {X 0,Y 124.401,Z 728.799,A -85,B 0,C 180,E1 -31140.235,E2 -31140.235} C_VEL
LIN {X 0,Y 121.755,Z 747.583,A -85,B 0,C 180,E1 -31140.517,E2 -31140.517} C_VEL
LIN {X 0,Y 118.334,Z 761.042,A -85,B 0,C 180,E1 -31140.728,E2 -31140.728} C_VEL
LIN {X 0,Y 118.009,Z 762.087,A -85,B 0,C 180,E1 -31140.748,E2 -31140.748} C_VEL
LIN {X 0,Y 117.907,Z 762.723,A -85,B 0,C 180,E1 -31140.757,E2 -31140.757} C_VEL
LIN {X 0,Y 117.907,Z 787.642,A -85,B 0,C 180,E1 -31140.757,E2 -31140.757} C_VEL
LIN {X 0,Y 109.441,Z 801.237,A -85,B 0,C 180,E1 -31140.814,E2 -31140.814} C_VEL
LIN {X 0,Y 100.975,Z 812.035,A -85,B 0,C 180,E1 -31140.88,E2 -31140.88} C_VEL
LIN {X 0,Y 89.415,Z 823.719,A -85,B 0,C 180,E1 -31140.991,E2 -31140.991} C_VEL
LIN {X 0,Y 77.856,Z 832.988,A -85,B 0,C 180,E1 -31141.134,E2 -31141.134} C_VEL
LIN {X 0,Y 67.625,Z 839.615,A -85,B 0,C 180,E1 -31141.302,E2 -31141.302} C_VEL
LIN {X 0,Y 65.932,Z 839.842,A -85,B 0,C 180,E1 -31141.335,E2 -31141.335} C_VEL
LIN {X 0,Y 60.521,Z 838.12,A -85,B 0,C 180,E1 -31141.452,E2 -31141.452} C_VEL
LIN {X 0,Y 59.127,Z 836.214,A -85,B 0,C 180,E1 -31141.486,E2 -31141.486} C_VEL
LIN {X 0,Y 59.127,Z 836.214,A -85,B 0,C 180,E1 -31141.486,E2 -31141.486} C_VEL
LIN {X 0,Y 56.257,Z 834.422,A -85,B 0,C 180,E1 -31141.809,E2 -31141.809} C_VEL
LIN {X 0,Y 45.766,Z 839.168,A -85,B 0,C 180,E1 -31143.357,E2 -31143.357} C_VEL
LIN {X 0,Y 35.337,Z 842.786,A -85,B 0,C 180,E1 -31145.972,E2 -31145.972} C_VEL
LIN {X 0,Y 28.448,Z 844.645,A -85,B 0,C 180,E1 -31148.749,E2 -31148.749} C_VEL
LIN {X 0,Y 21.657,Z 846.056,A -85,B 0,C 180,E1 -31153.148,E2 -31153.148} C_VEL
LIN {X 0,Y 9.12,Z 847.651,A -85,B 0,C 180,E1 -31179.534,E2 -31179.534} C_VEL
LIN {X 0,Y 5.967,Z 847.875,A -85,B 0,C 180,E1 -31229.944,E2 -31229.944} C_VEL
LIN {X 0,Y 9.076,Z 847.675,A -85,B 0,C 180,E1 -31280.684,E2 -31280.684} C_VEL
LIN {X 0,Y 21.645,Z 846.111,A -85,B 0,C 180,E1 -31306.856,E2 -31306.856} C_VEL
LIN {X 0,Y 28.434,Z 844.732,A -85,B 0,C 180,E1 -31311.289,E2 -31311.289} C_VEL
LIN {X 0,Y 38.262,Z 842.005,A -85,B 0,C 180,E1 -31315.023,E2 -31315.023} C_VEL
LIN {X 0,Y 40.81,Z 841.141,A -85,B 0,C 180,E1 -31317.669,E2 -31317.669} C_VEL
LIN {X 0,Y 41.103,Z 841.072,A -85,B 0,C 180,E1 -31320,E2 -31320} C_VEL
LIN {X 0,Y 35.21,Z 843.051,A -85,B 0,C 180,E1 -31323.785,E2 -31323.785} C_VEL
LIN {X 0,Y 28.269,Z 844.931,A -85,B 0,C 180,E1 -31326.159,E2 -31326.159} C_VEL
LIN {X 0,Y 21.422,Z 846.348,A -85,B 0,C 180,E1 -31330.288,E2 -31330.288} C_VEL
LIN {X 0,Y 8.813,Z 847.976,A -85,B 0,C 180,E1 -31357.18,E2 -31357.18} C_VEL
LIN {X 0,Y 5.895,Z 848.198,A -85,B 0,C 180,E1 -31410.057,E2 -31410.057} C_VEL
LIN {X 0,Y 8.822,Z 847.954,A -85,B 0,C 180,E1 -31462.87,E2 -31462.87} C_VEL
LIN {X 0,Y 21.432,Z 846.294,A -85,B 0,C 180,E1 -31489.748,E2 -31489.748} C_VEL
LIN {X 0,Y 28.278,Z 844.845,A -85,B 0,C 180,E1 -31493.894,E2 -31493.894} C_VEL
LIN {X 0,Y 38.705,Z 841.861,A -85,B 0,C 180,E1 -31497.205,E2 -31497.205} C_VEL
LIN {X 0,Y 49.207,Z 837.822,A -85,B 0,C 180,E1 -31499.134,E2 -31499.134} C_VEL
LIN {X 0,Y 56.229,Z 834.467,A -85,B 0,C 180,E1 -31500.148,E2 -31500.148} C_VEL
LIN {X 0,Y 56.257,Z 834.422,A -85,B 0,C 180,E1 -31501.809,E2 -31501.809} C_VEL
LIN {X 0,Y 56.257,Z 834.422,A -85,B 0,C 180,E1 -31501.809,E2 -31501.809}

QRS_NEXT_CUT()

QRS_NEXT()
QRS_HOME()

END
